{attribute 'strict'}
TYPE E_CR800StateDoingRequest :
(
	CR800_DOING_REQUEST_IDLE					:= 0,	(* DUMMY *)
	CR800_DOING_REQUEST_SEND_REQUEST			:= 10,	(* Send order reqest *)
	CR800_DOING_REQUEST_WAIT_FOR_CONFIRM		:= 20,	(* Wait for information that order is done *)
	CR800_DOING_REQUEST_DONE					:= 30	(* Request done *)
); 
END_TYPE

(* stored: Version 1.1.0.1, ProductVersion 3.1.4024.9
   DUT E_CR800StateDoingRequest: Id {ad459e6e-b97b-4320-9cb9-b62ad6c34760} *)
